PROGRAM MAIN
VAR
	fbTank : FB_TankController;
	fbHandle : FB_UpdateHandler;
END_VAR

fbTank();
fbHandle();

END_PROGRAM

(* stored: Version 1.1.0.1, ProductVersion 3.1.4024.16
   POU MAIN: Id {30ac5b1a-fc71-48d8-9064-af7f4cc0c250}, SpecialFunc None *)
